{attribute 'GeneratedUsingTerminal: EL3111-0000-0016'}
{attribute addProperty BoxType "EL3111-0000-0016"}
{attribute addProperty Id "AI_StandardAT %I*AI_Standard_A8DF64E310WcStateAT %I*WcState_9091E0EB2InfoDataAT %I*InfoData_94A18F5E2"}
{attribute addProperty CRC "306143992"}
{attribute addProperty Size "14"}
TYPE EL3111_123F62F8 EXTENDS EtcSlaveTerminalBase_947E5A46 :
STRUCT
	{attribute addProperty Name "AI_Standard"}
	AI_Standard : AI_Standard_A8DF64E3;
	{attribute addProperty Name "WcState"}
	WcState : WcState_9091E0EB;
	{attribute addProperty Name "InfoData"}
	InfoData : InfoData_94A18F5E;
END_STRUCT
END_TYPE

(* stored: Version 1.2.0.0, ProductVersion 3.1.4024.9
   DUT EL3111_123F62F8: Id {40fa4ecc-06d1-4adb-919d-05a8fbb6b24c} *)
